FUNCTION_BLOCK FB_ReloadRoundBeltBoxWithRobot_V2 EXTENDS FB_ObjectBase_V2 IMPLEMENTS IBasicElement
VAR_INPUT
    // Below are the components being controlled.
    Robot         : REFERENCE TO FB_FanucRobot_Basic_V2; // Fanuc Robot
    //AllocatedArea : REFERENCE TO FB_AllocatingSpace; // Allocated area , use to control round belt
	RoundBelt	: REFERENCE TO FB_RoundBeltService;
    WareHouse     : REFERENCE TO FB_WareHouse; // Storage area warehouse A and warehouse B conveyor and sensor
    //	A2_Sensor : REFERENCE TO FB_Sensor;
    //	A3_Sensor : REFERENCE TO FB_Sensor;
	Input : ST_InputTable;
    Info : ST_ReloadRoundBeltBox_Info; // Setting the feedin emptybox action's parameter
    Stop : BOOL;
END_VAR
VAR_OUTPUT
	AClampMoveDone	: BOOL;
	BClampMoveDone	: BOOL;
END_VAR
VAR
    strStatus         : STRING;
    tonTimeOut        : TON;
    tonFeedBoxTimeout : TON;
    _UniqueErrorCode  : STRING;
    PreviousStrStatus : STRING;
    PreviousErrorCode : STRING;
    A2_Sensor         : BOOL;
    A3_Sensor         : BOOL;
	//_Abort			  : BOOL;

	// Clamp work
	_AClampDoingWork	: BOOL;
	_BClampDoingWork	: BOOL;

	// ========== Resume 續做機制 ==========
	uiResumeStep	: UDINT := 0;	// 錯誤發生時記錄的步驟，供續做使用
	
	_bRetry			: BOOL;
END_VAR

SUPER^.A10_StateControl();
A00_BasicUnits();
A2_Sensor := Input.bRoundBelt_ChangeZoneA2Detect_Sensor;
A3_Sensor := Input.bRoundBelt_ChangeZoneA3Detect_Sensor;

(*============================================================
Create Date : 2025/11/22
Last Update	: 2026/03/31
Change Log  : 2025/11/24，send flag A clamp done and B clamp done for C# use to SQL // Owner : Gamin
			  2026/03/31，移植泰興鏡射版本，雷射續做，清除手臂錯誤。
============================================================*)

ACTION A00_BasicUnits:
tonTimeOut(PT:=T#60S);
tonFeedBoxTimeout(PT:=T#15s);
END_ACTION

METHOD M_CheckCommand : BOOL
VAR_INPUT
END_VAR
VAR_INST
	CheckBehavior : BOOL; // True :Behavior is correct
END_VAR
VAR
	I: INT;
END_VAR
// Memory clear
CheckBehavior := FALSE;
// Check command is correct
IF info.ClampA_Setting.Behavior = E_ClampWork.Work OR info.ClampB_Setting.Behavior = E_ClampWork.Work THEN
	CheckBehavior := TRUE;
ELSE
	CheckBehavior := FALSE;
END_IF


M_CheckCommand := CheckBehavior;
END_METHOD

METHOD M_CheckUnitsNotBusy : BOOL
VAR_INPUT
END_VAR
M_CheckUnitsNotBusy := true;
END_METHOD

METHOD M_CheckUnitsReady : BOOL
VAR_INPUT
END_VAR
M_CheckUnitsReady := true;
END_METHOD

METHOD M_SelectActionMode : E_ReloadRoundBoxAction
VAR_INPUT
END_VAR
IF info.ClampA_Setting.Behavior <> E_ClampWork.Work AND info.ClampB_Setting.Behavior <> E_ClampWork.Work THEN
	M_SelectActionMode :=E_ReloadRoundBoxAction.Undefined;
ELSIF info.ClampA_Setting.Behavior = E_ClampWork.Work AND info.ClampB_Setting.Behavior <> E_ClampWork.Work THEN
	IF info.ClampA_Setting.PickUpArea = E_ReloadRoundBelt_PickupArea.WareHouseA THEN
		M_SelectActionMode := E_ReloadRoundBoxAction.ClampA_WareHouseA;
	ELSIF info.ClampA_Setting.PickUpArea = E_ReloadRoundBelt_PickupArea.WareHouseB THEN
		M_SelectActionMode := E_ReloadRoundBoxAction.ClampA_WareHouseB;
	END_IF
ELSIF info.ClampA_Setting.Behavior <> E_ClampWork.Work AND info.ClampB_Setting.Behavior = E_ClampWork.Work THEN
	IF info.ClampB_Setting.PickUpArea = E_ReloadRoundBelt_PickupArea.WareHouseA THEN
		M_SelectActionMode := E_ReloadRoundBoxAction.ClampB_WareHouseA;
	ELSIF info.ClampB_Setting.PickUpArea = E_ReloadRoundBelt_PickupArea.WareHouseB THEN
		M_SelectActionMode := E_ReloadRoundBoxAction.ClampB_WareHouseB;
	END_IF
ELSIF info.ClampA_Setting.Behavior = E_ClampWork.Work AND info.ClampB_Setting.Behavior = E_ClampWork.Work THEN
	IF info.ClampA_Setting.PickUpArea = E_ReloadRoundBelt_PickupArea.WareHouseA THEN
		IF info.ClampB_Setting.PickUpArea = E_ReloadRoundBelt_PickupArea.WareHouseA THEN
			M_SelectActionMode := E_ReloadRoundBoxAction.A_WareHouseA_B_WareHouseA;
		ELSIF info.ClampB_Setting.PickUpArea = E_ReloadRoundBelt_PickupArea.WareHouseB THEN
			M_SelectActionMode := E_ReloadRoundBoxAction.A_WareHouseA_B_WareHouseB;
		END_IF
	ELSIF info.ClampA_Setting.PickUpArea = E_ReloadRoundBelt_PickupArea.WareHouseB THEN
		IF info.ClampB_Setting.PickUpArea = E_ReloadRoundBelt_PickupArea.WareHouseA THEN
			M_SelectActionMode := E_ReloadRoundBoxAction.A_WareHouseB_B_WareHouseA;
		ELSIF info.ClampB_Setting.PickUpArea = E_ReloadRoundBelt_PickupArea.WareHouseB THEN
			M_SelectActionMode := E_ReloadRoundBoxAction.A_WareHouseB_B_WareHouseB;
		END_IF
	END_IF
END_IF
END_METHOD

METHOD  M_STATE_ABORTED
VAR_INPUT
END_VAR
IF NOT _bRetry THEN
	Busy    := FALSE;
	Error	:= TRUE;
	Aborted := TRUE;
	_Abort  := TRUE;
	UniqueErrorCode := _UniqueErrorCode;
	Status := strStatus;
	_AbortCompleted := FALSE;
	uiAbortingStep	:= 0;
END_IF

IF Reset THEN
	_bRetry := TRUE;
	Error	:= FALSE;
	Aborted := FALSE;
	_Abort  := FALSE;
END_IF

// ============================================================
// Resume 機制：保持 Execute 並按 Reset 可從錯誤點繼續
// ============================================================
IF NOT Execute THEN
	eState := STATE_RESETTING;
ELSIF Execute AND _bRetry AND NOT Robot._DI1.Error AND NOT Robot.Halt THEN
	// Resume 模式：確認 Robot 不在暫停且無錯誤，從儲存的步驟繼續執行
	Status := '';

	uiExecutingStep := uiResumeStep;
	PreviousStrStatus := strStatus;
	PreviousErrorCode := _UniqueErrorCode;
	
	IF GVL_ADS.MachineState <>E_MachineState.Error THEN
		eSTATE:=STATE_EXECUTING;
	END_IF
END_IF
END_METHOD

METHOD  M_STATE_ABORTING
VAR_INPUT
END_VAR
CASE uiAbortingStep OF
	0:
			_Abort  := FALSE;
			_bRetry := FALSE;
			tonTimeOut.IN 		 := FALSE;
			tonFeedBoxTimeout.IN := FALSE;

			uiAbortingStep := 100;
	
    100:
			IF Robot._DI1.Error THEN
				uiAbortingStep := 200;
			ELSE
				uiAbortingStep := 9999;
			END_IF
	200:		
			 IF DAS_CoreSys.MachineControl.M_RobotResetCmd() THEN
				 uiAbortingStep := 300;
			 END_IF
	300:
			IF DAS_CoreSys.MachineControl.M_RobotStartCmd() THEN
				 uiAbortingStep := 400;
			 END_IF 
	400:
			IF Robot._DI1.Error THEN
		 		uiAbortingStep := 200;
			ELSE
				uiAbortingStep := 9999;
			END_IF
	9999:
			_AbortCompleted := TRUE;
END_CASE


IF _AbortCompleted THEN
    eState := STATE_Aborted;
END_IF
END_METHOD

METHOD  M_STATE_DONE
VAR_INPUT
END_VAR
Busy := FALSE;
Done := TRUE;
IF NOT Execute THEN
    eState := STATE_RESETTING;
END_IF
END_METHOD

METHOD  M_STATE_DORMANT
VAR_INPUT
END_VAR
// Clear FB output
Busy            := FALSE;
Done            := FALSE;
Aborted         := FALSE;
Error           := FALSE;
ErrorID         := 0;
Status          := '';
_ResetCompleted := FALSE;
_Error          := FALSE;
_Executed       := FALSE;
_Abort			:= FALSE;
uiExecutingStep := 0;
uiResettingStep := 0;
uiResumeStep    := 0;	// 清除 Resume 步驟
uiAbortingStep	:= 0;
tonTimeOut.IN := FALSE;
tonFeedBoxTimeout.IN := FALSE;
PreviousStrStatus := '';
PreviousErrorCode := '';
_UniqueErrorCode := '0';
AClampMoveDone := FALSE;
BClampMoveDone := FALSE;
_AClampDoingWork := FALSE;
_BClampDoingWork := FALSE;
_AbortCompleted	 := FALSE;
_bRetry			 := FALSE;

// Wait Execute command
IF Execute AND NOT stop THEN
    eState := STATE_EXECUTING;
END_IF
END_METHOD

METHOD  M_STATE_ERROR
VAR_INPUT
END_VAR
UniqueErrorCode	:= _UniqueErrorCode;
Error			:= TRUE;
status			:= strStatus;
Busy			:= FALSE;

IF NOT Execute THEN
    eState := STATE_RESETTING;
END_IF
END_METHOD

METHOD M_STATE_EXECUTING
VAR_INPUT
END_VAR
VAR_INST
    ActionMode       : E_ReloadRoundBoxAction;
	BoxReady_1st : BOOL;
	BoxReady_2nd : BOOL;
    CarrierReady_1st : BOOL;
    CarrierReady_2nd : BOOL;
    uiPickUpBothStep : UINT;
    uiPlaceBothStep  : UINT;
    ClampA_WareHouseCoordinates : ST_WareHouseCoordinates;
    ClampB_WareHouseCoordinates : ST_WareHouseCoordinates;
	
	//=============== test only====
		_A2Sensor	:BOOL;
		_A3Sensor	:BOOL;
END_VAR
// Set status busy
Busy := TRUE;
IF THIS^.Stop THEN // Pending the timeout when Stop signal occur
	tonTimeout.IN :=FALSE;
END_IF
CASE uiExecutingStep OF
    0:
        // Clear variable
        ActionMode       := E_ReloadRoundBoxAction.Undefined;
        CarrierReady_1st := FALSE;
        CarrierReady_2nd := FALSE;
        uiPickUpBothStep := 0;
        uiPlaceBothStep  := 0;
		BoxReady_1st := 0;
		BoxReady_2nd := 0;
        // Check command
        IF M_CheckCommand() THEN
            uiExecutingStep := 10;
        END_IF
    10:
        // Start process, check units first
        IF M_CheckUnitsReady() THEN
            uiExecutingStep := 20;
        END_IF
    20:
        // CHeck units not busy state
        IF M_CheckUnitsNotBusy() THEN
            uiExecutingStep := 1000;
        END_IF
    1000:
        // Select action mode
        ActionMode      := M_SelectActionMode();
        uiExecutingStep := 1100;
    1100:
		//DAS_CoreSys.MachineControl.fbAllocateArea.M_ActiveRoundBeltInternalCtrl(); //Request round belt 
		DAS_CoreSys.MachineControl.fbAllocateArea.M_GetRoundBeltAccess(ControlAccess := E_RoundBeltControlAccess.FanucRobot);
        CASE ActionMode OF
            E_ReloadRoundBoxAction.ClampA_WareHouseA:
                uiExecutingStep := 10000;
            E_ReloadRoundBoxAction.ClampA_WareHouseB:
                uiExecutingStep := 11000;
            E_ReloadRoundBoxAction.ClampB_WareHouseA:
                uiExecutingStep := 20000;
            E_ReloadRoundBoxAction.ClampB_WareHouseB:
                uiExecutingStep := 21000;
            E_ReloadRoundBoxAction.A_WareHouseA_B_WareHouseA:
                uiExecutingStep := 30000;
            E_ReloadRoundBoxAction.A_WareHouseA_B_WareHouseB:
                uiExecutingStep := 31000;
            E_ReloadRoundBoxAction.A_WareHouseB_B_WareHouseA:
                uiExecutingStep := 32000;
            E_ReloadRoundBoxAction.A_WareHouseB_B_WareHouseB:
                uiExecutingStep := 33000;
        END_CASE
    10000: // Only ClampA pickup box from WarehouseA
        IF NOT Robot._DI1.Done THEN
            // Read ClampA Warehouse coordinate
            ClampA_WareHouseCoordinates := info.ClampA_Setting.WareHouseSetting;
            // Reload Warehouse target position box
            WareHouse.M_StartReloadBox(WareHouseSelect := E_WareHouse.WareHouseA, WarehouseCoordinates := ClampA_WareHouseCoordinates);

            // Check Box reload completed
            IF WareHouse.bReloadBox_Completed THEN
                BoxReady_1st 	 := TRUE;
				_AClampDoingWork := TRUE;
            END_IF

            // Robot Warehouse move
            Robot.M_StartWareHousePickUpBox_ClampA(WareHouseSelect := E_WareHouse.WareHouseA,
                                                   Info            := ClampA_WareHouseCoordinates,
                                                   BoxReady_1st    := BoxReady_1st);

            DAS_CoreSys.MachineControl.fbAllocateArea.M_GetRoundBeltAccess(ControlAccess := E_RoundBeltControlAccess.FanucRobot);
            DAS_CoreSys.MachineControl.fbAllocateArea.M_StartReloadRoundBeltAtion(ReloadStation := info.ClampA_Setting.RoundBeltSetting.Station);
			
			// make sure robot doing AClamp done
			IF _AClampDoingWork AND  NOT Robot._DI1.ClampA_Open THEN
				AClampMoveDone := TRUE;
			END_IF
        ELSE
			tonTimeOut.IN :=FALSE;
            uiExecutingStep := 10080;
        END_IF
		tonTimeOut.IN :=TRUE;
		IF tonTimeOut.Q THEN
			uiResumeStep := 10000;
			_Abort := TRUE;
			tonTimeOut.IN :=FALSE;
			strStatus :='FB_ReloadRoundBeltBoxWithRobot_V2 Step 10000: Pick Box timeout';
		END_IF
    10080:
        Robot.M_ResetAllCommand(); // Clear command and go to place box
		WareHouse.M_ResetReloadBox();
        IF NOT Robot._DI1.Done THEN
            uiExecutingStep := 60000; // only place clampA
        END_IF
    11000: // Only ClampA pickup box from WarehouseB
        IF NOT Robot._DI1.Done THEN
            // Read ClampA Warehouse coordinate
            ClampA_WareHouseCoordinates := info.ClampA_Setting.WareHouseSetting;
            // Reload Warehouse target position box
            WareHouse.M_StartReloadBox(WareHouseSelect := E_WareHouse.WareHouseB, WarehouseCoordinates := ClampA_WareHouseCoordinates);

            // Check Box reload completed
            IF WareHouse.bReloadBox_Completed THEN
                BoxReady_1st 	 := TRUE;
				_AClampDoingWork := TRUE;
            END_IF

            // Robot Warehouse move
            Robot.M_StartWareHousePickUpBox_ClampA(WareHouseSelect := E_WareHouse.WareHouseB,
                                                   Info            := ClampA_WareHouseCoordinates,
                                                   BoxReady_1st    := BoxReady_1st);

            DAS_CoreSys.MachineControl.fbAllocateArea.M_GetRoundBeltAccess(ControlAccess := E_RoundBeltControlAccess.FanucRobot);
            DAS_CoreSys.MachineControl.fbAllocateArea.M_StartReloadRoundBeltAtion(ReloadStation := info.ClampA_Setting.RoundBeltSetting.Station);
			
			// make sure robot doing AClamp done
			IF _AClampDoingWork AND  NOT Robot._DI1.ClampA_Open THEN
				AClampMoveDone := TRUE;
			END_IF

        ELSE
			tonTimeOut.IN :=FALSE;
            uiExecutingStep := 11080;
        END_IF
		tonTimeOut.IN :=TRUE;
		IF tonTimeOut.Q THEN
			uiResumeStep := 11000;
			_Abort := TRUE;
			tonTimeOut.IN :=FALSE;
			strStatus :='FB_ReloadRoundBeltBoxWithRobot_V2 Step 11000: Pick Box timeout';
		END_IF
    11080:
        Robot.M_ResetAllCommand(); // Clear command and go to place box

        IF NOT Robot._DI1.Done THEN
            uiExecutingStep := 60000; // only place clampA
        END_IF
    20000: // Only ClampB pickup from WarehouseA
        IF NOT Robot._DI1.Done THEN
            // Read ClampA Warehouse coordinate
            ClampB_WareHouseCoordinates := info.ClampB_Setting.WareHouseSetting;
            // Reload Warehouse target position box
            WareHouse.M_StartReloadBox(WareHouseSelect := E_WareHouse.WareHouseA, WarehouseCoordinates := ClampB_WareHouseCoordinates);

            // Check Box reload completed
            IF WareHouse.bReloadBox_Completed THEN
                BoxReady_2nd 	 := TRUE;
				_BClampDoingWork := TRUE;
            END_IF

            // Robot Warehouse move
            Robot.M_StartWareHousePickUpBox_ClampB(WareHouseSelect := E_WareHouse.WareHouseA,
                                                   Info            := ClampB_WareHouseCoordinates,
                                                   BoxReady_2nd    := BoxReady_2nd);

          	DAS_CoreSys.MachineControl.fbAllocateArea.M_GetRoundBeltAccess(ControlAccess := E_RoundBeltControlAccess.FanucRobot);
            DAS_CoreSys.MachineControl.fbAllocateArea.M_StartReloadRoundBeltAtion(ReloadStation := info.ClampB_Setting.RoundBeltSetting.Station);
			
			// robot doing BClamp done
			IF _BClampDoingWork AND NOT Robot._DI1.ClampB_Open THEN 
				BClampMoveDone := TRUE;
			END_IF

        ELSE
			tonTimeOut.IN :=FALSE;
            uiExecutingStep := 20080;
        END_IF
			tonTimeOut.IN :=TRUE;
		IF tonTimeOut.Q THEN
			uiResumeStep := 20000;
			_Abort := TRUE;
			tonTimeOut.IN :=FALSE;
			strStatus :='FB_ReloadRoundBeltBoxWithRobot_V2 Step 20000: Pick Box timeout';
		END_IF
    20080:
        WareHouse.M_ResetReloadBox();
        Robot.M_ResetAllCommand();

        IF NOT Robot._DI1.Done THEN
            uiExecutingStep := 70000; // Only ClampB place box
        END_IF
    21000: // Only ClampB pickup from WarehouseB
        IF NOT Robot._DI1.Done THEN
            // Read ClampA Warehouse coordinate
            ClampB_WareHouseCoordinates := info.ClampB_Setting.WareHouseSetting;
            // Reload Warehouse target position box
            WareHouse.M_StartReloadBox(WareHouseSelect := E_WareHouse.WareHouseB, WarehouseCoordinates := ClampB_WareHouseCoordinates);

            // Check Box reload completed
            IF WareHouse.bReloadBox_Completed THEN
                BoxReady_2nd 	 := TRUE;
				_BClampDoingWork := TRUE;
            END_IF

            // Robot Warehouse move
            Robot.M_StartWareHousePickUpBox_ClampB(WareHouseSelect := E_WareHouse.WareHouseB,
                                                   Info            := ClampB_WareHouseCoordinates,
                                                   BoxReady_2nd    := BoxReady_2nd);
            DAS_CoreSys.MachineControl.fbAllocateArea.M_GetRoundBeltAccess(ControlAccess := E_RoundBeltControlAccess.FanucRobot);
            DAS_CoreSys.MachineControl.fbAllocateArea.M_StartReloadRoundBeltAtion(ReloadStation := info.ClampA_Setting.RoundBeltSetting.Station);
			
			// robot doing BClamp done
			IF _BClampDoingWork AND NOT Robot._DI1.ClampB_Open THEN 
				BClampMoveDone := TRUE;
			END_IF

        ELSE
			tonTimeOut.IN :=FALSE;
            uiExecutingStep := 21080;
        END_IF
			tonTimeOut.IN :=TRUE;
		IF tonTimeOut.Q THEN
			uiResumeStep := 21000;
			_Abort := TRUE;
			tonTimeOut.IN :=FALSE;
			strStatus :='FB_ReloadRoundBeltBoxWithRobot_V2 Step 21000: Pick Box timeout';
		END_IF
    21080:
        WareHouse.M_ResetReloadBox();
        Robot.M_ResetAllCommand();

        IF NOT Robot._DI1.Done THEN
            uiExecutingStep := 70000; // Only ClampB place box
        END_IF
    30000: // ClampA and ClampB pickup box from WarehouseA
        ClampA_WareHouseCoordinates := info.ClampA_Setting.WareHouseSetting;
        ClampB_WareHouseCoordinates := info.ClampB_Setting.WareHouseSetting;

        CASE uiPickUpBothStep OF
            0: // ClampA target slide move the box to front side
                WareHouse.M_StartReloadBox(WareHouseSelect      := E_WareHouse.WareHouseA,
                                           WarehouseCoordinates := ClampA_WareHouseCoordinates);

              	DAS_CoreSys.MachineControl.fbAllocateArea.M_GetRoundBeltAccess(ControlAccess := E_RoundBeltControlAccess.FanucRobot);
                DAS_CoreSys.MachineControl.fbAllocateArea.M_StartReloadRoundBeltAtion(ReloadStation := info.ClampA_Setting.RoundBeltSetting.Station);

                IF WareHouse.bReloadBox_Completed THEN
                    BoxReady_1st     := TRUE;
					_AClampDoingWork := TRUE;
                    uiPickUpBothStep := 10;
                END_IF

            10: // wait Robot Allow continue
                IF Robot._DI1.Notification AND
                    NOT
                    WareHouse._stWarehouseList.ASide_Layers[ClampA_WareHouseCoordinates.Layer].stStatus.bSlides[ClampA_WareHouseCoordinates.Slide]
                    THEN
                    WareHouse.M_ResetReloadBox();

                    IF NOT WareHouse.bReloadBox_Completed THEN
                        uiPickUpBothStep := 20;
                    END_IF

                END_IF
            20: // ClampB target slide move the box to front slide
                WareHouse.M_StartReloadBox(WareHouseSelect := E_WareHouse.WareHouseA, WarehouseCoordinates := ClampB_WareHouseCoordinates);

                IF WareHouse.bReloadBox_Completed THEN
                    BoxReady_2nd     := TRUE;
					_BClampDoingWork := TRUE;
                    uiPickUpBothStep := 99;
                END_IF
            99:
        // wait reset
        END_CASE

        Robot.M_StartWareHousePickUpBox_ClampBoth(WareHouseSelect := E_WareHouse.WareHouseA,
                                                  ClampA_Info     := ClampA_WareHouseCoordinates,
                                                  ClampB_Info     := ClampB_WareHouseCoordinates,
                                                  BoxReady_1st    := BoxReady_1st,
                                                  BoxReady_2nd    := BoxReady_2nd);
												  
		// robot doing AClamp done
			IF _AClampDoingWork AND  NOT Robot._DI1.ClampA_Open THEN
				AClampMoveDone := TRUE;
			END_IF

		// robot doing BClamp done
			IF _BClampDoingWork AND NOT Robot._DI1.ClampB_Open THEN 
				BClampMoveDone := TRUE;
			END_IF										  

        IF Robot._DI1.Done THEN
			tonTimeOut.IN :=FALSE;
            uiExecutingStep := 30080;
        END_IF
			tonTimeOut.IN :=TRUE;
		IF tonTimeOut.Q THEN
			uiResumeStep := 30000;
			_Abort := TRUE;
			tonTimeOut.IN :=FALSE;
			strStatus :='FB_ReloadRoundBeltBoxWithRobot_V2 Step 30000: Pick Box timeout';
		END_IF
    30080: // Check robot command is clear
        WareHouse.M_ResetReloadBox();
        Robot.M_ResetAllCommand();

        IF NOT Robot._DI1.Done THEN
            uiExecutingStep := 80000; // go to place step
        END_IF
    31000: // ClampA pickup from Warehouse A, ClampB pickup from Warehouse B
        IF NOT Robot._DI1.Done THEN
            ClampA_WareHouseCoordinates := info.ClampA_Setting.WareHouseSetting;
            WareHouse.M_StartReloadBox(WareHouseSelect := E_WareHouse.WareHouseA, WarehouseCoordinates := ClampA_WareHouseCoordinates);

            IF WareHouse.bReloadBox_Completed THEN
                BoxReady_1st     := TRUE;
				_AClampDoingWork := TRUE;
            END_IF
			DAS_CoreSys.MachineControl.fbAllocateArea.M_ActiveRoundBeltInternalCtrl();
			DAS_CoreSys.MachineControl.fbAllocateArea.M_StartReloadRoundBeltAtion(ReloadStation := info.ClampA_Setting.RoundBeltSetting.Station);
            Robot.M_StartWareHousePickUpBox_ClampA(WareHouseSelect := E_WareHouse.WareHouseA,
                                                   Info            := ClampA_WareHouseCoordinates,
                                                   BoxReady_1st    := BoxReady_1st);
			
			// robot doing AClamp done
			IF _AClampDoingWork AND  NOT Robot._DI1.ClampA_Open THEN
				AClampMoveDone := TRUE;
			END_IF						   
												   
        ELSE
			tonTimeOut.IN :=FALSE;
            uiExecutingStep := 31080;
        END_IF
			tonTimeOut.IN :=TRUE;
		IF tonTimeOut.Q THEN
			uiResumeStep := 31000;
			_Abort := TRUE;
			tonTimeOut.IN :=FALSE;
			strStatus :='FB_ReloadRoundBeltBoxWithRobot_V2 Step 31000: Pick Box timeout';
		END_IF

    31080:
        Robot.M_ResetAllCommand(); // Clear command and go to place box
		WareHouse.M_ResetReloadBox();
        IF NOT Robot._di1.Done THEN
            uiExecutingStep := 31100; // ClampA pickup finished, ClampB pickup start
        END_IF
    31100:
        IF NOT Robot._di1.Done THEN
            ClampB_WareHouseCoordinates := info.ClampB_Setting.WareHouseSetting;
            WareHouse.M_StartReloadBox(WareHouseSelect := E_WareHouse.WareHouseB, WarehouseCoordinates := ClampB_WareHouseCoordinates);

            IF WareHouse.bReloadBox_Completed THEN
                BoxReady_2nd 	 := TRUE;
				_BClampDoingWork := TRUE;
            END_IF

            Robot.M_StartWareHousePickUpBox_ClampB(WareHouseSelect := E_WareHouse.WareHouseB,
                                                   Info            := ClampB_WareHouseCoordinates,
                                                   BoxReady_2nd    := BoxReady_2nd);
												   
			// robot doing BClamp done
			IF _BClampDoingWork AND NOT Robot._DI1.ClampB_Open THEN 
				BClampMoveDone := TRUE;
			END_IF
												   
        ELSE
			tonTimeOut.IN :=FALSE;
            uiExecutingStep := 31180;
        END_IF
				tonTimeOut.IN :=TRUE;
		IF tonTimeOut.Q THEN
			uiResumeStep := 31100;
			_Abort := TRUE;
			tonTimeOut.IN :=FALSE;
			strStatus :='FB_ReloadRoundBeltBoxWithRobot_V2 Step 31100: Pick Box timeout';
		END_IF
    31180:
        Robot.M_ResetAllCommand(); // Clear command and go to place box

        IF NOT Robot._DI1.Done THEN
            uiExecutingStep := 80000; // only place clampA
        END_IF
    32000: // CLampA pickup from Warehouse B, ClampB pickup from Warehouse A
        IF NOT Robot._DI1.Done THEN
            ClampA_WareHouseCoordinates := info.ClampA_Setting.WareHouseSetting;
            WareHouse.M_StartReloadBox(WareHouseSelect := E_WareHouse.WareHouseB, WarehouseCoordinates := ClampA_WareHouseCoordinates);

            IF WareHouse.bReloadBox_Completed THEN
                BoxReady_1st 	 := TRUE;
				_AClampDoingWork := TRUE;
            END_IF
            DAS_CoreSys.MachineControl.fbAllocateArea.M_GetRoundBeltAccess(ControlAccess := E_RoundBeltControlAccess.FanucRobot);
            DAS_CoreSys.MachineControl.fbAllocateArea.M_StartReloadRoundBeltAtion(ReloadStation := info.ClampA_Setting.RoundBeltSetting.Station);
            Robot.M_StartWareHousePickUpBox_ClampA(WareHouseSelect := E_WareHouse.WareHouseB,
                                                   Info            := ClampA_WareHouseCoordinates,
                                                   BoxReady_1st    := BoxReady_1st);
												   
			// robot doing AClamp done
			IF _AClampDoingWork AND  NOT Robot._DI1.ClampA_Open THEN
				AClampMoveDone := TRUE;
			END_IF									   
												   
        ELSE
			tonTimeOut.IN :=FALSE;
            uiExecutingStep := 32080;
        END_IF
				tonTimeOut.IN :=TRUE;
		IF tonTimeOut.Q THEN
			uiResumeStep := 32000;
			_Abort := TRUE;
			tonTimeOut.IN :=FALSE;
			strStatus :='FB_ReloadRoundBeltBoxWithRobot_V2 Step 32000: Pick Box timeout';
		END_IF

    32080:
        Robot.M_ResetAllCommand(); // Clear command and go to place box
		WareHouse.M_ResetReloadBox();
        IF NOT Robot._di1.Done THEN
            uiExecutingStep := 32100; // ClampA pickup finished, ClampB pickup start
        END_IF
    32100:
        IF NOT Robot._di1.Done THEN
            ClampB_WareHouseCoordinates := info.ClampB_Setting.WareHouseSetting;
            WareHouse.M_StartReloadBox(WareHouseSelect := E_WareHouse.WareHouseA, WarehouseCoordinates := ClampB_WareHouseCoordinates);

            IF WareHouse.bReloadBox_Completed THEN
                BoxReady_2nd 	 := TRUE;
				_BClampDoingWork := TRUE;
            END_IF

            Robot.M_StartWareHousePickUpBox_ClampB(WareHouseSelect := E_WareHouse.WareHouseA,
                                                   Info            := ClampB_WareHouseCoordinates,
                                                   BoxReady_2nd    := BoxReady_2nd);
												   
			// robot doing BClamp done
			IF _BClampDoingWork AND NOT Robot._DI1.ClampB_Open THEN 
				BClampMoveDone := TRUE;
			END_IF									   
												   
        ELSE
			tonTimeOut.IN :=FALSE;
            uiExecutingStep := 32180;
        END_IF
				tonTimeOut.IN :=TRUE;
		IF tonTimeOut.Q THEN
			uiResumeStep := 32100;
			_Abort := TRUE;
			tonTimeOut.IN :=FALSE;
			strStatus :='FB_ReloadRoundBeltBoxWithRobot_V2 Step 32100: Pick Box timeout';
		END_IF

    32180:
        Robot.M_ResetAllCommand(); // Clear command and go to place box
		WareHouse.M_ResetReloadBox();
        IF NOT Robot._DI1.Done THEN
            uiExecutingStep := 80000; // only place clampA
        END_IF
    33000: // Both Clamp pickup from WarehouseB
        ClampA_WareHouseCoordinates := info.ClampA_Setting.WareHouseSetting;
        ClampB_WareHouseCoordinates := info.ClampB_Setting.WareHouseSetting;

        CASE uiPickUpBothStep OF
            0: // ClampA target slide move the box to front side
                WareHouse.M_StartReloadBox(WareHouseSelect      := E_WareHouse.WareHouseB,
                                           WarehouseCoordinates := ClampA_WareHouseCoordinates);

                DAS_CoreSys.MachineControl.fbAllocateArea.M_GetRoundBeltAccess(ControlAccess := E_RoundBeltControlAccess.FanucRobot );
                DAS_CoreSys.MachineControl.fbAllocateArea.M_StartReloadRoundBeltAtion(ReloadStation := info.ClampA_Setting.RoundBeltSetting.Station);

                IF WareHouse.bReloadBox_Completed THEN
                    BoxReady_1st     := TRUE;
					_AClampDoingWork := TRUE;
                    uiPickUpBothStep := 10;
                END_IF

            10: // wait Robot Allow continue
                IF Robot._DI1.Notification AND
                    NOT
                    WareHouse._stWarehouseList.BSide_Layers[ClampA_WareHouseCoordinates.Layer].stStatus.bSlides[ClampA_WareHouseCoordinates.Slide]
                    THEN
                    WareHouse.M_ResetReloadBox();

                    IF NOT WareHouse.bReloadBox_Completed THEN
                        uiPickUpBothStep := 20;
                    END_IF

                END_IF
            20: // ClampB target slide move the box to front slide
                WareHouse.M_StartReloadBox(WareHouseSelect := E_WareHouse.WareHouseB, WarehouseCoordinates := ClampB_WareHouseCoordinates);

                IF WareHouse.bReloadBox_Completed THEN
                    BoxReady_2nd     := TRUE;
					_BClampDoingWork := TRUE;
                    uiPickUpBothStep := 99;
                END_IF
            99:
        // wait reset
        END_CASE

        Robot.M_StartWareHousePickUpBox_ClampBoth(WareHouseSelect := E_WareHouse.WareHouseB,
                                                  ClampA_Info     := ClampA_WareHouseCoordinates,
                                                  ClampB_Info     := ClampB_WareHouseCoordinates,
                                                  BoxReady_1st    := BoxReady_1st,
                                                  BoxReady_2nd    := BoxReady_2nd);
												  
		// robot doing AClamp done
			IF _AClampDoingWork AND  NOT Robot._DI1.ClampA_Open THEN
				AClampMoveDone := TRUE;
			END_IF

		// robot doing BClamp done
			IF _BClampDoingWork AND NOT Robot._DI1.ClampB_Open THEN 
				BClampMoveDone := TRUE;
			END_IF										  
												  

        IF Robot._DI1.Done THEN
			tonTimeOut.IN :=FALSE;
            uiExecutingStep := 33080;
        END_IF
		
			tonTimeOut.IN :=TRUE;
		IF tonTimeOut.Q THEN
			uiResumeStep := 33000;
			_Abort := TRUE;
			tonTimeOut.IN :=FALSE;
			strStatus :='FB_ReloadRoundBeltBoxWithRobot_V2 Step 33000: Pick Box timeout';
		END_IF

    33080:
        WareHouse.M_ResetReloadBox();
        Robot.M_ResetAllCommand();

        IF NOT Robot._DI1.Done THEN
            uiExecutingStep := 80000;
        END_IF
    60000: // Only ClampA place box
        WareHouse.M_ResetReloadBox();
        Robot.M_ResetAllCommand();

        // Check Robot RSR1 not working
        IF NOT Robot._di1.Done AND
            NOT (Robot._DI1.AbsMoveA OR
            Robot._DI1.AbsMoveB OR
            Robot._DI1.WarehouseA OR
            Robot._DI1.WarehouseB) THEN
			DAS_CoreSys.MachineControl.fbAllocateArea.M_GetRoundBeltAccess(ControlAccess := E_RoundBeltControlAccess.FanucRobot);
            uiExecutingStep := 61000;
        END_IF
    61000:
        
				DAS_CoreSys.MachineControl.fbAllocateArea.M_GetRoundBeltAccess(ControlAccess := E_RoundBeltControlAccess.FanucRobot);
				DAS_CoreSys.MachineControl.fbAllocateArea.M_StartReloadRoundBeltAtion(ReloadStation := info.ClampA_Setting.RoundBeltSetting.Station);
				IF RoundBelt.xDone  AND arAxisCtrl_gb[AxisNo.RoundBelt].Admin.Axis.Status.NotMoving THEN	
					DAS_CoreSys.MachineControl.fbAllocateArea.M_ResetReloadRoundBeltAction();	
					CarrierReady_1st:=TRUE;			
				 	uiExecutingStep := 61010;
			    END_IF
				IF RoundBelt.xError THEN
					_Error :=TRUE;
					DAS_CoreSys.MachineControl.fbAllocateArea.M_ResetReloadRoundBeltAction();	
					strStatus:='FB_ReloadRoundBeltBoxWithRobot_V2 Step 61000: RoundBelt Error';
				END_IF
	61010:
			
        IF NOT Robot._DI1.Done THEN
            Robot.M_StartMoveBoxToRoundBelt_ClampA(CarrierSelect := info.ClampA_Setting.RoundBeltSetting.ReloadCarrier,
                                                   A2_Sensor     := A2_Sensor,
                                                   A3_Sensor     := A3_Sensor,
                                                   RoundBeltSafe := CarrierReady_1st);
        ELSE
			tonTimeOut.IN :=FALSE;
            uiExecutingStep := 61080;
        END_IF
			tonTimeOut.IN :=TRUE;
		IF tonTimeOut.Q THEN
			uiResumeStep := 61010;
			_Abort := TRUE;
			tonTimeOut.IN :=FALSE;
			strStatus :='FB_ReloadRoundBeltBoxWithRobot_V2 Step 61010: Place Box timeout';
		END_IF
		IF Robot._DI1.Error THEN
			uiResumeStep := 61010;
			_Abort := TRUE;
			strStatus :=CONCAT(STR1 := 'FB_ReloadRoundBeltBoxWithRobot_V2 Step 61010: ',
							   STR2 := Robot.ErrMsg);
		END_IF

    61080:
		DAS_CoreSys.MachineControl.fbAllocateArea.M_ResetReloadRoundBeltAction();
        DAS_CoreSys.MachineControl.fbAllocateArea.M_ReleaseRoundBeltAccess(ControlAccess := E_RoundBeltControlAccess.FanucRobot);
        Robot.M_ResetAllCommand();

        IF NOT Robot._DI1.Done THEN
            uiExecutingStep := 99000; // Go to process end
        END_IF
    70000: // Only ClampB place box
        WareHouse.M_ResetReloadBox();
        Robot.M_ResetAllCommand();

        // Check Robot RSR1 not working
        IF NOT Robot._di1.Done AND
            NOT (Robot._DI1.AbsMoveA OR
            Robot._DI1.AbsMoveB OR
            Robot._DI1.WarehouseA OR
            Robot._DI1.WarehouseB) THEN
            uiExecutingStep := 71000;
        END_IF
    71000:
        // Active RoundBelt INTERNAL control
//               DAS_CoreSys.MachineControl.fbAllocateArea.M_GetRoundBeltAccess(ControlAccess := E_RoundBeltControlAccess.FanucRobot);
//               DAS_CoreSys.MachineControl.fbAllocateArea.M_StartReloadRoundBeltAtion(ReloadStation := info.ClampB_Setting.RoundBeltSetting.Station);
				IF RoundBelt.xDone THEN
					DAS_CoreSys.MachineControl.fbAllocateArea.M_ResetReloadRoundBeltAction();
					//DAS_CoreSys.MachineControl.fbAllocateArea.M_ReleaseRoundBeltAccess(ControlAccess := E_RoundBeltControlAccess.FanucRobot);
					CarrierReady_2nd :=TRUE;
				 	uiExecutingStep := 71010;
			    END_IF
				IF RoundBelt.xError THEN
					_Error :=TRUE;
					DAS_CoreSys.MachineControl.fbAllocateArea.M_ResetReloadRoundBeltAction();
					DAS_CoreSys.MachineControl.fbAllocateArea.M_ReleaseRoundBeltAccess(ControlAccess := E_RoundBeltControlAccess.FanucRobot);
					strStatus:='FB_ReloadRoundBeltBoxWithRobot_V2 Step 71000: RoundBelt Error';
				END_IF
	71010:
			
        IF NOT Robot._DI1.Done THEN
            Robot.M_StartMoveBoxToRoundBelt_ClampB(CarrierSelect := info.ClampB_Setting.RoundBeltSetting.ReloadCarrier,
                                                   A2_Sensor     := A2_Sensor,
                                                   A3_Sensor     := A3_Sensor,
                                                   RoundBeltSafe := CarrierReady_2nd);
        ELSE
			tonTimeOut.IN :=FALSE;
            uiExecutingStep := 71080;
        END_IF
			tonTimeOut.IN :=TRUE;
		IF tonTimeOut.Q THEN
			uiResumeStep := 71010;
			_Abort := TRUE;
			tonTimeOut.IN :=FALSE;
			strStatus :='FB_ReloadRoundBeltBoxWithRobot_V2 Step 71010: Place Box timeout';
		END_IF
		IF Robot._DI1.Error THEN
			uiResumeStep := 71010;
			_Abort := TRUE;
			strStatus :=CONCAT(STR1 := 'FB_ReloadRoundBeltBoxWithRobot_V2 Step 71010: ',
							   STR2 := Robot.ErrMsg);
		END_IF

    71080:
		DAS_CoreSys.MachineControl.fbAllocateArea.M_ResetReloadRoundBeltAction();
        DAS_CoreSys.MachineControl.fbAllocateArea.M_ReleaseRoundBeltAccess(ControlAccess :=E_RoundBeltControlAccess.FanucRobot );       
        Robot.M_ResetAllCommand();

        IF NOT Robot._DI1.Done THEN
            uiExecutingStep := 99000; // Go to process end
        END_IF
    80000:                            // Both Clamp place box
        WareHouse.M_ResetReloadBox(); // Clear Warehouse reload command
        Robot.M_ResetAllCommand();    // Clear Fanuc Robot command
        IF NOT Robot._DI1.Done THEN
            uiExecutingStep := 81000;
        END_IF;
    81000:
        CASE uiPlaceBothStep OF
            0:
				//=============
				_A2Sensor:=FALSE;
				_A3Sensor:=FALSE;
				//==============
                CarrierReady_1st := FALSE;
                CarrierReady_2nd := FALSE;
				DAS_CoreSys.MachineControl.fbAllocateArea.M_GetRoundBeltAccess(ControlAccess := E_RoundBeltControlAccess.FanucRobot);
                uiPlaceBothStep  := 10;
            10:
                // Check move Round Belt done
                IF RoundBelt.xDone THEN
					DAS_CoreSys.MachineControl.fbAllocateArea.M_ResetReloadRoundBeltAction();
					DAS_CoreSys.MachineControl.fbAllocateArea.M_ReleaseRoundBeltAccess(ControlAccess :=E_RoundBeltControlAccess.FanucRobot );       
                    CarrierReady_1st := TRUE;
                    uiPlaceBothStep  := 11;
                END_IF
				IF RoundBelt.xError THEN
					_Error :=TRUE;
					DAS_CoreSys.MachineControl.fbAllocateArea.M_ResetReloadRoundBeltAction();
					DAS_CoreSys.MachineControl.fbAllocateArea.M_ReleaseRoundBeltAccess(ControlAccess :=E_RoundBeltControlAccess.FanucRobot );       
					strStatus:='FB_ReloadRoundBeltBoxWithRobot_V2 Step 81000: RoundBelt Error';
				END_IF
            11:
				//========================Test==================
				IF info.ClampA_Setting.RoundBeltSetting.ReloadCarrier = E_ReloadRoundBelt_PlaceAddress.A2 AND NOT A2_Sensor THEN
					_A2Sensor		:= A2_Sensor;
					uiPlaceBothStep := 15;
				ELSIF info.ClampA_Setting.RoundBeltSetting.ReloadCarrier = E_ReloadRoundBelt_PlaceAddress.A2 AND  A2_Sensor THEN				//edited By Gamin 2026/04/02，放盒位有盒就報警
					_Abort 	  := TRUE;
					strStatus := 'FB_ReloadRoundBeltBoxWithRobot_V2 Step 81000: ClampA place A2 Position has box';
				END_IF
				IF info.ClampA_Setting.RoundBeltSetting.ReloadCarrier = E_ReloadRoundBelt_PlaceAddress.A3 AND NOT A3_Sensor THEN
					_A3Sensor		:= A3_Sensor;
					uiPlaceBothStep := 15;
				ELSIF info.ClampA_Setting.RoundBeltSetting.ReloadCarrier = E_ReloadRoundBelt_PlaceAddress.A3 AND  A3_Sensor THEN
					_Abort	  := TRUE;
					strStatus := 'FB_ReloadRoundBeltBoxWithRobot_V2 Step 81000: ClampA place A3 Position has box'; 
				END_IF
				
			15:
				//======================End_test==================
                IF ((info.ClampA_Setting.RoundBeltSetting.ReloadCarrier = E_ReloadRoundBelt_PlaceAddress.A2) AND A2_Sensor) OR
                    ((info.ClampA_Setting.RoundBeltSetting.ReloadCarrier = E_ReloadRoundBelt_PlaceAddress.A3) AND A3_Sensor)
                    THEN
					DAS_CoreSys.MachineControl.fbAllocateArea.M_GetRoundBeltAccess(ControlAccess := E_RoundBeltControlAccess.FanucRobot);
                    uiPlaceBothStep :=20;// 30;
                END_IF
            20:
                // Wait Notification
                IF robot._DI1.Notification THEN
					//========================Test==================
						IF info.ClampA_Setting.RoundBeltSetting.ReloadCarrier = E_ReloadRoundBelt_PlaceAddress.A2 THEN
							_A2Sensor:=FALSE;
						END_IF
						IF info.ClampA_Setting.RoundBeltSetting.ReloadCarrier = E_ReloadRoundBelt_PlaceAddress.A3 THEN
							_A3Sensor:=FALSE;
						END_IF
				//======================End_test==================
                    DAS_CoreSys.MachineControl.fbAllocateArea.M_ResetReloadRoundBeltAction();

                    IF NOT RoundBelt.xDone THEN
                        uiPlaceBothStep := 30;
                    END_IF
                END_IF
            30: // Move Round belt 2nd time
				DAS_CoreSys.MachineControl.fbAllocateArea.M_GetRoundBeltAccess(ControlAccess := E_RoundBeltControlAccess.FanucRobot);
				DAS_CoreSys.MachineControl.fbAllocateArea.M_StartReloadRoundBeltAtion(ReloadStation := info.ClampB_Setting.RoundBeltSetting.Station);
                uiPlaceBothStep := 40;
            40:
                IF RoundBelt.xDone THEN
					DAS_CoreSys.MachineControl.fbAllocateArea.M_ResetReloadRoundBeltAction();
                    CarrierReady_2nd := TRUE;
                    uiPlaceBothStep  := 80;
                END_IF
				IF RoundBelt.xError THEN
					_Error :=TRUE;
					DAS_CoreSys.MachineControl.fbAllocateArea.M_ResetReloadRoundBeltAction();	
					strStatus:='FB_ReloadRoundBeltBoxWithRobot_V2 Step 81000: RoundBelt Error';
				END_IF
            80:	
				//========================Test==================
				IF info.ClampB_Setting.RoundBeltSetting.ReloadCarrier = E_ReloadRoundBelt_PlaceAddress.A2 AND NOT A2_Sensor THEN
					_A2Sensor:=A2_Sensor;
					uiPlaceBothStep := 99;
				ELSIF info.ClampB_Setting.RoundBeltSetting.ReloadCarrier = E_ReloadRoundBelt_PlaceAddress.A2 AND  A2_Sensor THEN
					_Abort	  := TRUE;
					strStatus := 'FB_ReloadRoundBeltBoxWithRobot_V2 Step 81000: ClampB place A2 Position has box'; 
				END_IF
				IF info.ClampB_Setting.RoundBeltSetting.ReloadCarrier = E_ReloadRoundBelt_PlaceAddress.A3 AND NOT A3_Sensor THEN
					_A3Sensor:=A3_Sensor;
					uiPlaceBothStep := 99;
				ELSIF info.ClampB_Setting.RoundBeltSetting.ReloadCarrier = E_ReloadRoundBelt_PlaceAddress.A3 AND  A3_Sensor THEN
					_Abort	  := TRUE;
					strStatus := 'FB_ReloadRoundBeltBoxWithRobot_V2 Step 81000: ClampB place A3 Position has box'; 
				END_IF
				//======================End_test==================
			99:
				;
			
        // wait reset
        END_CASE

        IF NOT Robot._DI1.Done THEN
            Robot.M_StartMoveBoxToRoundBelt_Both(CarrierSelect_ClampA := info.ClampA_Setting.RoundBeltSetting.ReloadCarrier,
                                                 CarrierSelect_ClampB := info.ClampB_Setting.RoundBeltSetting.ReloadCarrier,
                                                 A2_Sensor            := _A2Sensor,//A2_Sensor,
                                                 A3_Sensor            := _A3Sensor,//A3_Sensor,
                                                 RoundBeltSafe_1st    := CarrierReady_1st,
                                                 RoundBeltSafe_2nd    := CarrierReady_2nd);
        ELSE
			tonTimeOut.IN :=FALSE;
            uiExecutingStep := 99000;
        END_IF
			tonTimeOut.IN :=TRUE;
		IF tonTimeOut.Q THEN
			uiResumeStep := 81000;
			_Abort := TRUE;
			tonTimeOut.IN :=FALSE;
			strStatus :='FB_ReloadRoundBeltBoxWithRobot_V2 Step 81000: Place Box timeout';
		END_IF
		IF Robot._DI1.Error THEN
			uiResumeStep := 81000;
			_Abort		 := TRUE;
			strStatus	 := CONCAT(STR1 := 'FB_ReloadRoundBeltBoxWithRobot_V2 Step 81000: ',
								   STR2 := Robot.ErrMsg);
		END_IF
		
    99000: // process done

			DAS_CoreSys.MachineControl.fbAllocateArea.M_ResetReloadRoundBeltAction();
			DAS_CoreSys.MachineControl.fbAllocateArea.M_ReleaseRoundBeltAccess(ControlAccess :=E_RoundBeltControlAccess.FanucRobot );       
        	Status    := 'FB_ReloadRoundBeltBoxWithRobot_V2 Step 99000: Process completed';
        	_Executed := TRUE;
END_CASE

IF _Executed THEN
    eState := STATE_DONE;
ELSIF NOT Execute THEN
    eState := STATE_RESETTING;
ELSIF Abort OR _Abort THEN
	eState :=STATE_ABORTING;
ELSIF _Error THEN
	eState :=STATE_ERROR;
END_IF
END_METHOD

METHOD  M_STATE_RESETTING
VAR_INPUT
END_VAR
IF _Executed THEN Done :=TRUE; END_IF

CASE uiResettingStep OF
	0:
		AClampMoveDone	:= FALSE;
		BClampMoveDone	:= FALSE;
		_AClampDoingWork	:= FALSE;
		_BClampDoingWork	:= FALSE;
		DAS_CoreSys.MachineControl.fbAllocateArea.M_ResetReloadRoundBeltAction();
		DAS_CoreSys.MachineControl.fbAllocateArea.M_ReleaseRoundBeltAccess(ControlAccess :=E_RoundBeltControlAccess.FanucRobot );       
		WareHouse.M_ResetReloadBox();
		Robot.M_ResetAllCommand();
		uiResettingStep := 100;
	100:
		_ResetCompleted := TRUE;
END_CASE
IF _ResetCompleted THEN
    eState := STATE_DORMANT;
END_IF
END_METHOD

END_FUNCTION_BLOCK

(* stored: Version 1.1.0.1, ProductVersion 3.1.4024.13
   POU FB_ReloadRoundBeltBoxWithRobot_V2: Id {f8136e28-b84a-4612-a381-3bb5c569a57e}, SpecialFunc None
   Folder Method: Id {7846ed69-ca7c-44e3-8239-25dc73879ab8}
   Folder State: Id {cd922701-f9b7-465b-a413-35e59b046456}
   Action A00_BasicUnits: Id {f97d9ee0-90c4-429a-983f-769c6674e7dd}
   Method M_CheckCommand: Id {546ea1d9-b4fb-432e-8839-c84cf3ab0c4b}
   Method M_CheckUnitsNotBusy: Id {5fad0094-95d4-4d01-a28c-72bf1014ff95}
   Method M_CheckUnitsReady: Id {c32d0f78-51c0-4817-a42a-ae5b9778d51b}
   Method M_SelectActionMode: Id {ba5d5b67-4790-472c-a57f-228b082f5cb3}
   Method M_STATE_ABORTED: Id {75bba4ee-b93b-47a1-b2f6-ab4fa8844dc4}
   Method M_STATE_ABORTING: Id {7831b399-cdc2-43a9-a280-2b6ae5d62bd9}
   Method M_STATE_DONE: Id {2dcc9306-8daf-42c4-972d-01a8153741f4}
   Method M_STATE_DORMANT: Id {41eb431a-ec91-411c-b6a4-d797c75cfcfc}
   Method M_STATE_ERROR: Id {9e67305c-9bc9-4a5c-a7b3-cddb256782aa}
   Method M_STATE_EXECUTING: Id {48ee86ae-68c0-4c53-91f0-704d5e08d084}
   Method M_STATE_RESETTING: Id {5cb52fc3-bd9e-4796-9423-533bb02a4f78} *)
